// Mitsubishi GX Works2 project: 三菱步进电机控制   PLC: FX1S

PROGRAM MAIN
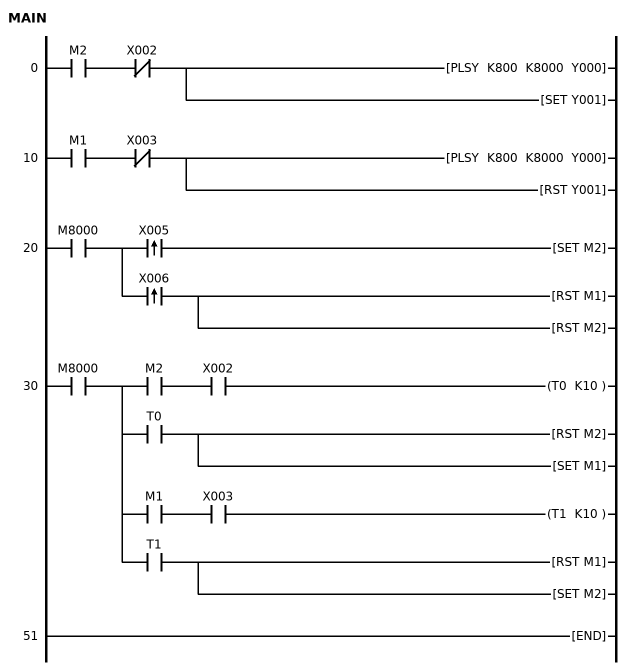
0     LD      M2
      ANI     X002
      PLSY    K800 K8000 Y000
      SET     Y001
10    LD      M1
      ANI     X003
      PLSY    K800 K8000 Y000
      RST     Y001
20    LD      M8000
      MPS
      ANDP    X005
      SET     M2
      MPP
      ANDP    X006
      RST     M1
      RST     M2
30    LD      M8000
      MPS
      AND     M2
      AND     X002
      OUT     T0 K10
      MRD
      AND     T0
      RST     M2
      SET     M1
      MRD
      AND     M1
      AND     X003
      OUT     T1 K10
      MPP
      AND     T1
      RST     M1
      SET     M2
51    END
END_PROGRAM
